Staubli VAL3: object.dtx

public num nID
public trsf trTrsf
public num nLatchedValue
